PROGRAM p_ALI
VAR
	fbALI_A	:	FB_ALI;
END_VAR

END_PROGRAM

(* stored: Version 1.1.0.1, ProductVersion 3.1.4020.12
   POU p_ALI: Id {2f24df4a-4e55-4a2a-b530-4a66a8831e7d}, SpecialFunc None *)
